{attribute 'GeneratedUsingTerminal: EL5151-0000-0016'}
{attribute addProperty BoxType "EL5151-0000-0016"}
{attribute addProperty Id "Period_valueAT %I*UDINT4"}
{attribute addProperty CRC "615922771"}
{attribute addProperty Size "4"}
TYPE ENC_Inputs_24B63C53 :
STRUCT
	{attribute addProperty Name "Period_value"}
	Period_value AT %I* : UDINT;
END_STRUCT
END_TYPE

(* stored: Version 1.2.0.0, ProductVersion 3.1.4024.9
   DUT ENC_Inputs_24B63C53: Id {8e356e27-c045-4a84-996e-efc12eb8cc63} *)
